Yaskawa INFORM job: blower_planes_program.JBI

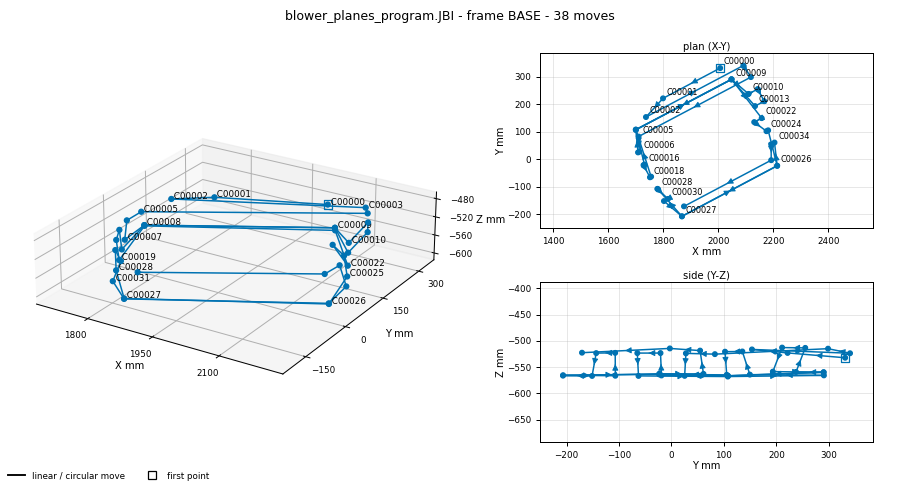
[picture p0: tool path of blower_planes_program.JBI in frame BASE, 38 of 40 moves have a stored position in this frame; points joined in program order, loops and branches not executed]
/JOB
//NAME blower_planes_program
//POS
///NPOS 38,0,38,0,0,0
///TOOL 0
///POSTYPE BASE
///RECTAN
///RCONF 0,0,0,0,0,0,0,0,0,0,0,0,0,0,0,0,0,0,0,0,0,0,0,0
C00000=2007.344125,331.194468,-532.168850,175.000000,-5.000000,5.000000
C00001=1799.935034,221.412893,-522.933777,175.000000,-5.000000,5.000000
C00002=1738.041780,153.510261,-516.274777,175.000000,-5.000000,5.000000
C00003=2091.314362,340.497342,-523.558777,175.000000,-5.000000,5.000000
C00004=2118.926047,298.540161,-514.829777,175.000000,-5.000000,5.000000
C00005=1711.308596,82.788356,-525.288777,175.000000,-5.000000,5.000000
C00006=1713.803633,27.536940,-523.756777,175.000000,-5.000000,5.000000
C00007=1709.266248,25.135304,-566.645282,175.000000,-45.614216,27.892257
C00008=1701.142604,107.624185,-566.675292,175.000000,-45.625885,-17.127802
C00009=2048.357023,290.173307,-559.901082,-175.000000,-44.770103,-107.088038
C00010=2110.468187,237.491380,-559.185872,-175.000000,-44.385784,-152.107743
C00011=2143.735111,255.099554,-513.325777,175.000000,5.000000,5.000000
C00012=2167.239644,210.968458,-512.757777,175.000000,-5.000000,5.000000
C00013=2133.869848,193.305834,-558.587949,-175.000000,-44.396202,-152.107743
C00014=2048.379268,290.168112,-559.775451,-175.000000,-44.771373,-107.101785
C00015=1701.131295,107.595873,-566.457457,175.000000,-45.624879,-17.112274
C00016=1732.666109,-19.051194,-565.920849,175.000000,-45.603798,27.892257
C00017=1729.175172,-20.898946,-523.205777,175.000000,5.000000,5.000000
C00018=1752.479959,-65.135767,-523.247777,175.000000,-5.000000,5.000000
C00019=1756.737026,-62.882503,-566.768874,175.000000,-45.203468,27.892257
C00020=1701.670017,107.439810,-568.013008,175.000000,-45.342038,-17.110418
C00021=2048.664770,290.663967,-565.759969,175.000000,-45.054168,-107.111452
C00022=2158.005186,149.508624,-564.297601,175.000000,-44.796532,-152.107743
C00023=2130.899682,135.161688,-520.206777,175.000000,5.000000,5.000000
C00024=2175.380567,102.133370,-520.567777,175.000000,-5.000000,5.000000
C00025=2181.504950,105.375005,-564.730134,175.000000,-44.857483,-152.107743
C00026=2214.337022,-23.355453,-563.908135,175.000000,-44.701021,162.889260
C00027=1868.546491,-206.659253,-565.483346,-175.000000,-44.902565,72.887704
C00028=1780.227783,-107.020890,-566.461153,-175.000000,-45.142517,27.892257
C00029=1779.731926,-107.283346,-522.794777,175.000000,5.000000,5.000000
C00030=1818.112182,-143.540726,-523.284777,175.000000,-5.000000,5.000000
C00031=1803.329789,-151.365042,-566.805446,175.000000,-45.322129,27.892257
C00032=1868.497828,-206.889157,-566.220081,175.000000,-45.030580,72.893724
C00033=2214.086766,-23.289260,-562.656023,-175.000000,-44.573083,162.887021
C00034=2204.579808,61.016483,-562.893092,-175.000000,-44.677871,-152.107743
C00035=2192.475838,54.609854,-518.521777,175.000000,5.000000,5.000000
C00036=2192.528931,-3.088151,-514.364777,175.000000,-5.000000,5.000000
C00037=1876.077101,-170.586018,-522.512777,175.000000,-5.000000,5.000000
///POSTYPE PULSE
///PULSE
EC00000=120832.0
EC00001=120832.0
EC00002=120832.0
EC00003=120832.0
EC00004=120832.0
EC00005=120832.0
EC00006=120832.0
EC00007=120832.0
EC00008=120832.0
EC00009=120832.0
EC00010=120832.0
EC00011=120832.0
EC00012=120832.0
EC00013=120832.0
EC00014=120832.0
EC00015=120832.0
EC00016=120832.0
EC00017=120832.0
EC00018=120832.0
EC00019=120832.0
EC00020=120832.0
EC00021=120832.0
EC00022=120832.0
EC00023=120832.0
EC00024=120832.0
EC00025=120832.0
EC00026=120832.0
EC00027=120832.0
EC00028=120832.0
EC00029=120832.0
EC00030=120832.0
EC00031=120832.0
EC00032=120832.0
EC00033=120832.0
EC00034=120832.0
EC00035=120832.0
EC00036=120832.0
EC00037=120832.0
//INST
///DATE 2023/08/16 15:41
///ATTR SC,RW,RJ
////FRAME BASE
///GROUP1 RB1,ST1
NOP
MOVJ P009 EX000 VJ=15.00
MOVJ C00000 EC00000 VJ=15.0
CALL JOB:SPYON
MOVL C00001 EC00001 V=150.0
MOVL C00002 EC00002 V=150.0
MOVL C00003 EC00003 V=150.0
MOVL C00004 EC00004 V=150.0
MOVL C00005 EC00005 V=150.0
MOVL C00006 EC00006 V=150.0
MOVL C00007 EC00007 V=150.0
MOVL C00008 EC00008 V=150.0
MOVL C00009 EC00009 V=150.0
MOVL C00010 EC00010 V=150.0
MOVL C00011 EC00011 V=150.0
MOVL C00012 EC00012 V=150.0
MOVL C00013 EC00013 V=150.0
MOVL C00014 EC00014 V=150.0
MOVL C00015 EC00015 V=150.0
MOVL C00016 EC00016 V=150.0
MOVL C00017 EC00017 V=150.0
MOVL C00018 EC00018 V=150.0
MOVL C00019 EC00019 V=150.0
MOVL C00020 EC00020 V=150.0
MOVL C00021 EC00021 V=150.0
MOVL C00022 EC00022 V=150.0
MOVL C00023 EC00023 V=150.0
MOVL C00024 EC00024 V=150.0
MOVL C00025 EC00025 V=150.0
MOVL C00026 EC00026 V=150.0
MOVL C00027 EC00027 V=150.0
MOVL C00028 EC00028 V=150.0
MOVL C00029 EC00029 V=150.0
MOVL C00030 EC00030 V=150.0
MOVL C00031 EC00031 V=150.0
MOVL C00032 EC00032 V=150.0
MOVL C00033 EC00033 V=150.0
MOVL C00034 EC00034 V=150.0
MOVL C00035 EC00035 V=150.0
MOVL C00036 EC00036 V=150.0
MOVL C00037 EC00037 V=150.0
CALL JOB:SPYOF
MOVJ P009 VJ=15.00
END
